FUNCTION_BLOCK State_Levi_Pullup_and_Dropdown
VAR_INPUT
	configured_peak_current: LREAL;
	current : LREAL;
END_VAR

VAR_OUTPUT
	force_values : ARRAY[0..11] OF INT;
END_VAR

VAR
	count_cycles: INT;
END_VAR

	force_values[0] := LREAL_TO_INT((current * 1000.0)/ configured_peak_current);
	force_values[1] := LREAL_TO_INT((current * 1000.0)/ configured_peak_current);
	
	force_values[2] := LREAL_TO_INT((current * 1000.0)/ configured_peak_current);
	force_values[3] := LREAL_TO_INT((current * 1000.0)/ configured_peak_current);
	
	force_values[4] := LREAL_TO_INT((current * 1000.0)/ configured_peak_current);
	force_values[5] := LREAL_TO_INT((current * 1000.0)/ configured_peak_current);
	
	force_values[6] := LREAL_TO_INT((current * 1000.0)/ configured_peak_current);
	force_values[7] := LREAL_TO_INT((current * 1000.0)/ configured_peak_current);
	
	force_values[8] := 0;
	force_values[9] := 0;
	
	force_values[10] := 0;
	force_values[11] := 0;
	
	count_cycles := count_cycles + 1;
	
	IF count_cycles > 1000 THEN
		count_cycles := 0;
	END_IF

END_FUNCTION_BLOCK

(* stored: Version 1.1.0.1
   POU State_Levi_Pullup_and_Dropdown: Id {a8ff25ca-1bdd-4e92-a06b-7bf324690b4b}, SpecialFunc None *)
